// SIMATIC S7-200 SMART project (STEP 7-Micro/WIN SMART), CPU ST40

SYMBOL_TABLE Table 1
FWD_Timer        T102
REV_Timer        T101
REV              Q0.1
FWD              Q0.0
FWD_Memory       M0.2
REV_Memory       M0.1
Memory_1         M0.0
Sensor           I0.2
Stop_SW          I0.1
Start_SW         I0.0
END_SYMBOL_TABLE

ORGANIZATION_BLOCK MAIN:OB1
TITLE=Program Comments
BEGIN
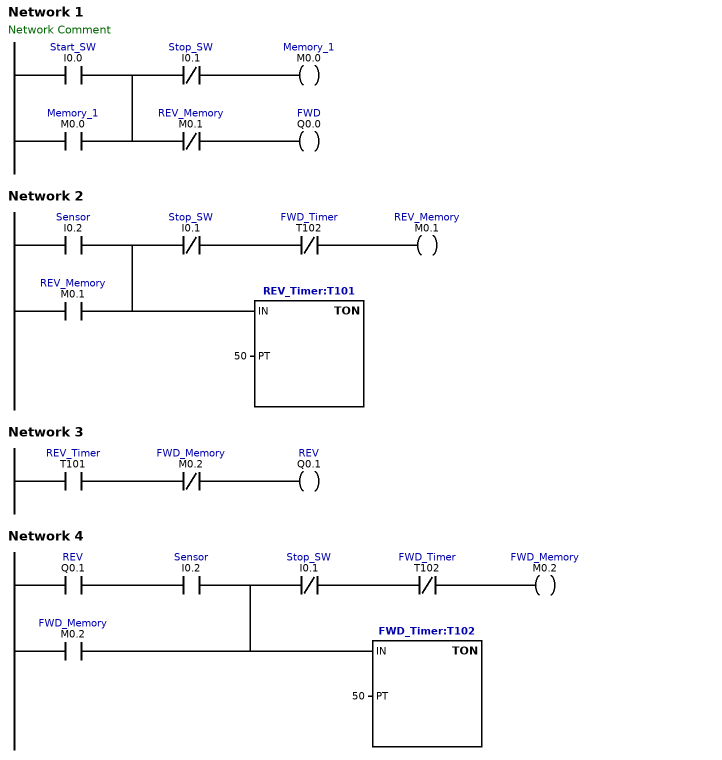
Network 1
// Network Comment
LD     Start_SW:I0.0
O      Memory_1:M0.0
LPS
AN     Stop_SW:I0.1
=      Memory_1:M0.0
LPP
AN     REV_Memory:M0.1
=      FWD:Q0.0
Network 2
LD     Sensor:I0.2
O      REV_Memory:M0.1
LPS
AN     Stop_SW:I0.1
AN     FWD_Timer:T102
=      REV_Memory:M0.1
LPP
TON    REV_Timer:T101, 50
Network 3
LD     REV_Timer:T101
AN     FWD_Memory:M0.2
=      REV:Q0.1
Network 4
LD     REV:Q0.1
A      Sensor:I0.2
O      FWD_Memory:M0.2
LPS
AN     Stop_SW:I0.1
AN     FWD_Timer:T102
=      FWD_Memory:M0.2
LPP
TON    FWD_Timer:T102, 50
END_ORGANIZATION_BLOCK
